PROGRAM MAIN
VAR
	fb05D100 : IO.FB_O5D100;
END_VAR

fb05D100();

END_PROGRAM

(* stored: Version 1.1.0.1, ProductVersion 3.1.4024.12
   POU MAIN: Id {851d153b-ef72-434d-b1dc-408dc36f46e2}, SpecialFunc None *)
